// TIA Portal V17 export
// export: Created 2024-06-14T09:52:43.5267752Z, ExportSetting WithDefaults, DisplayName Totally Integrated Automation Portal, DisplayVersion V17, DisplayName TIA Portal Openness, DisplayVersion V17, DisplayName TIA Portal Version Control Interface, DisplayVersion V17, DisplayName Simotion SCOUT TIA, DisplayVersion 5.4.3.0, DisplayName SINAMICS Startdrive Advanced, DisplayVersion V17 SP1 Update 1, DisplayName SINAMICS Startdrive G110M, G120, G120C, G120D, G120P, G115D, DisplayVersion V17 SP1 Update 1, DisplayName SINAMICS Startdrive G130, G150, S120, S150, SINAMICS MV, S210, DisplayVersion V17 SP1 Update 1, DisplayName STEP 7 Professional, DisplayVersion V17, DisplayName STEP 7 Safety, DisplayVersion V17, DisplayName WinCC Professional, DisplayVersion V17
DATA_BLOCK "MOD_TCP_SETUP_DB"   // DB100
{ S7_Optimized_Access := 'FALSE' }
VERSION : 0.1
// stored: AutoNumber false, DBAccessibleFromOPCUA true, IsOnlyStoredInLoadMemory false, IsWriteProtectedInAS false
   VAR RETAIN
      TCP_Data_Station4 { ExternalAccessible := 'False'; ExternalVisible := 'False'; ExternalWritable := 'False'; S7_SetPoint := 'True'} : Array[1..6] of "Mod_TCP_Data";
      TCP_Data_Station5 { ExternalAccessible := 'False'; ExternalVisible := 'False'; ExternalWritable := 'False'} : Array[1..6] of "Mod_TCP_Data";
      TCP_Data_CHECK_SCALE_1 { S7_SetPoint := 'True'} : "Mod_TCP_Data";
      TCP_Data_CORRECTION_SCALE { S7_SetPoint := 'True'} : "Mod_TCP_Data";
   END_VAR
BEGIN
   TCP_Data_Station4[1..6].Mod_TCP_Connect.connectParamClient.InterfaceId := 64;
   TCP_Data_Station4[1].Mod_TCP_Connect.connectParamClient.ID := 1;
   TCP_Data_Station4[2].Mod_TCP_Connect.connectParamClient.ID := 2;
   TCP_Data_Station4[3].Mod_TCP_Connect.connectParamClient.ID := 3;
   TCP_Data_Station4[4].Mod_TCP_Connect.connectParamClient.ID := 4;
   TCP_Data_Station4[5].Mod_TCP_Connect.connectParamClient.ID := 5;
   TCP_Data_Station4[6].Mod_TCP_Connect.connectParamClient.ID := 6;
   TCP_Data_Station4[1..6].Mod_TCP_Connect.connectParamClient.ConnectionType := 16#0B;
   TCP_Data_Station4[1..6].Mod_TCP_Connect.connectParamClient.ActiveEstablished := true;
   TCP_Data_Station4[1].Mod_TCP_Connect.connectParamClient.RemoteAddress.ADDR[1] := 192;
   TCP_Data_Station4[1].Mod_TCP_Connect.connectParamClient.RemoteAddress.ADDR[2] := 168;
   TCP_Data_Station4[1].Mod_TCP_Connect.connectParamClient.RemoteAddress.ADDR[3] := 0;
   TCP_Data_Station4[1].Mod_TCP_Connect.connectParamClient.RemoteAddress.ADDR[4] := 21;
   TCP_Data_Station4[2].Mod_TCP_Connect.connectParamClient.RemoteAddress.ADDR[1] := 192;
   TCP_Data_Station4[2].Mod_TCP_Connect.connectParamClient.RemoteAddress.ADDR[2] := 168;
   TCP_Data_Station4[2].Mod_TCP_Connect.connectParamClient.RemoteAddress.ADDR[3] := 0;
   TCP_Data_Station4[2].Mod_TCP_Connect.connectParamClient.RemoteAddress.ADDR[4] := 22;
   TCP_Data_Station4[3].Mod_TCP_Connect.connectParamClient.RemoteAddress.ADDR[1] := 192;
   TCP_Data_Station4[3].Mod_TCP_Connect.connectParamClient.RemoteAddress.ADDR[2] := 168;
   TCP_Data_Station4[3].Mod_TCP_Connect.connectParamClient.RemoteAddress.ADDR[3] := 0;
   TCP_Data_Station4[3].Mod_TCP_Connect.connectParamClient.RemoteAddress.ADDR[4] := 23;
   TCP_Data_Station4[4].Mod_TCP_Connect.connectParamClient.RemoteAddress.ADDR[1] := 192;
   TCP_Data_Station4[4].Mod_TCP_Connect.connectParamClient.RemoteAddress.ADDR[2] := 168;
   TCP_Data_Station4[4].Mod_TCP_Connect.connectParamClient.RemoteAddress.ADDR[3] := 0;
   TCP_Data_Station4[4].Mod_TCP_Connect.connectParamClient.RemoteAddress.ADDR[4] := 24;
   TCP_Data_Station4[5].Mod_TCP_Connect.connectParamClient.RemoteAddress.ADDR[1] := 192;
   TCP_Data_Station4[5].Mod_TCP_Connect.connectParamClient.RemoteAddress.ADDR[2] := 168;
   TCP_Data_Station4[5].Mod_TCP_Connect.connectParamClient.RemoteAddress.ADDR[3] := 0;
   TCP_Data_Station4[5].Mod_TCP_Connect.connectParamClient.RemoteAddress.ADDR[4] := 25;
   TCP_Data_Station4[6].Mod_TCP_Connect.connectParamClient.RemoteAddress.ADDR[1] := 192;
   TCP_Data_Station4[6].Mod_TCP_Connect.connectParamClient.RemoteAddress.ADDR[2] := 168;
   TCP_Data_Station4[6].Mod_TCP_Connect.connectParamClient.RemoteAddress.ADDR[3] := 0;
   TCP_Data_Station4[6].Mod_TCP_Connect.connectParamClient.RemoteAddress.ADDR[4] := 26;
   TCP_Data_Station4[1..6].Mod_TCP_Connect.connectParamClient.RemotePort := 502;
   TCP_Data_Station4[2..6].Mod_TCP_Connect.connectParamClient.LocalPort := 0;
   TCP_Data_Station4[1].Mod_Client[1..6].request := false;
   TCP_Data_Station4[2].Mod_Client[1..6].request := false;
   TCP_Data_Station4[3].Mod_Client[1..6].request := false;
   TCP_Data_Station4[4].Mod_Client[1..6].request := false;
   TCP_Data_Station4[5].Mod_Client[1..6].request := false;
   TCP_Data_Station4[6].Mod_Client[1..6].request := false;
   TCP_Data_Station4[1].Mod_Client[1..6].enable := false;
   TCP_Data_Station4[2].Mod_Client[1..6].enable := false;
   TCP_Data_Station4[3].Mod_Client[1..6].enable := false;
   TCP_Data_Station4[4].Mod_Client[1..6].enable := false;
   TCP_Data_Station4[5].Mod_Client[1..6].enable := false;
   TCP_Data_Station4[6].Mod_Client[1..6].enable := false;
   TCP_Data_Station4[1].Mod_Client[1..6].disconnect := false;
   TCP_Data_Station4[2].Mod_Client[1..6].disconnect := false;
   TCP_Data_Station4[3].Mod_Client[1..6].disconnect := false;
   TCP_Data_Station4[4].Mod_Client[1..6].disconnect := false;
   TCP_Data_Station4[5].Mod_Client[1..6].disconnect := false;
   TCP_Data_Station4[6].Mod_Client[1..6].disconnect := false;
   TCP_Data_Station4[1].Mod_Client[1..6].done := false;
   TCP_Data_Station4[2].Mod_Client[1..6].done := false;
   TCP_Data_Station4[3].Mod_Client[1..6].done := false;
   TCP_Data_Station4[4].Mod_Client[1..6].done := false;
   TCP_Data_Station4[5].Mod_Client[1..6].done := false;
   TCP_Data_Station4[6].Mod_Client[1..6].done := false;
   TCP_Data_Station4[1].Mod_Client[1..6].busy := false;
   TCP_Data_Station4[2].Mod_Client[1..6].busy := false;
   TCP_Data_Station4[3].Mod_Client[1..6].busy := false;
   TCP_Data_Station4[4].Mod_Client[1..6].busy := false;
   TCP_Data_Station4[5].Mod_Client[1..6].busy := false;
   TCP_Data_Station4[6].Mod_Client[1..6].busy := false;
   TCP_Data_Station4[1].Mod_Client[1..6].error := false;
   TCP_Data_Station4[2].Mod_Client[1..6].error := false;
   TCP_Data_Station4[3].Mod_Client[1..6].error := false;
   TCP_Data_Station4[4].Mod_Client[1..6].error := false;
   TCP_Data_Station4[5].Mod_Client[1..6].error := false;
   TCP_Data_Station4[6].Mod_Client[1..6].error := false;
   TCP_Data_Station4[1].Mod_Client[1..6].status := 16#0;
   TCP_Data_Station4[2].Mod_Client[1..6].status := 16#0;
   TCP_Data_Station4[3].Mod_Client[1..6].status := 16#0;
   TCP_Data_Station4[4].Mod_Client[1..6].status := 16#0;
   TCP_Data_Station4[5].Mod_Client[1..6].status := 16#0;
   TCP_Data_Station4[6].Mod_Client[1..6].status := 16#0;
   TCP_Data_Station4[1].Mod_Client[1..6].statusSave := 16#0;
   TCP_Data_Station4[2].Mod_Client[1..6].statusSave := 16#0;
   TCP_Data_Station4[3].Mod_Client[1..6].statusSave := 16#0;
   TCP_Data_Station4[4].Mod_Client[1..6].statusSave := 16#0;
   TCP_Data_Station4[5].Mod_Client[1..6].statusSave := 16#0;
   TCP_Data_Station4[6].Mod_Client[1..6].statusSave := 16#0;
   TCP_Data_Station4[1].Mod_Client[1].modbusMode := 1;
   TCP_Data_Station4[1].Mod_Client[2].modbusMode := 0;
   TCP_Data_Station4[1].Mod_Client[3].modbusMode := 1;
   TCP_Data_Station4[1].Mod_Client[4..5].modbusMode := 0;
   TCP_Data_Station4[1].Mod_Client[6].modbusMode := 1;
   TCP_Data_Station4[2].Mod_Client[1].modbusMode := 1;
   TCP_Data_Station4[2].Mod_Client[2].modbusMode := 0;
   TCP_Data_Station4[2].Mod_Client[3].modbusMode := 1;
   TCP_Data_Station4[2].Mod_Client[4..5].modbusMode := 0;
   TCP_Data_Station4[2].Mod_Client[6].modbusMode := 1;
   TCP_Data_Station4[3].Mod_Client[1].modbusMode := 1;
   TCP_Data_Station4[3].Mod_Client[2].modbusMode := 0;
   TCP_Data_Station4[3].Mod_Client[3].modbusMode := 1;
   TCP_Data_Station4[3].Mod_Client[4..5].modbusMode := 0;
   TCP_Data_Station4[3].Mod_Client[6].modbusMode := 1;
   TCP_Data_Station4[4].Mod_Client[1].modbusMode := 1;
   TCP_Data_Station4[4].Mod_Client[2].modbusMode := 0;
   TCP_Data_Station4[4].Mod_Client[3].modbusMode := 1;
   TCP_Data_Station4[4].Mod_Client[4..5].modbusMode := 0;
   TCP_Data_Station4[4].Mod_Client[6].modbusMode := 1;
   TCP_Data_Station4[5].Mod_Client[1].modbusMode := 1;
   TCP_Data_Station4[5].Mod_Client[2].modbusMode := 0;
   TCP_Data_Station4[5].Mod_Client[3].modbusMode := 1;
   TCP_Data_Station4[5].Mod_Client[4..5].modbusMode := 0;
   TCP_Data_Station4[5].Mod_Client[6].modbusMode := 1;
   TCP_Data_Station4[6].Mod_Client[1].modbusMode := 1;
   TCP_Data_Station4[6].Mod_Client[2].modbusMode := 0;
   TCP_Data_Station4[6].Mod_Client[3].modbusMode := 1;
   TCP_Data_Station4[6].Mod_Client[4..5].modbusMode := 0;
   TCP_Data_Station4[6].Mod_Client[6].modbusMode := 1;
   TCP_Data_Station4[1].Mod_Client[1].modbusDataAddress := 40908;
   TCP_Data_Station4[1].Mod_Client[2].modbusDataAddress := 40001;
   TCP_Data_Station4[1].Mod_Client[3].modbusDataAddress := 40302;
   TCP_Data_Station4[1].Mod_Client[4].modbusDataAddress := 0;
   TCP_Data_Station4[1].Mod_Client[5].modbusDataAddress := 1;
   TCP_Data_Station4[1].Mod_Client[6].modbusDataAddress := 0;
   TCP_Data_Station4[2].Mod_Client[1].modbusDataAddress := 40908;
   TCP_Data_Station4[2].Mod_Client[2].modbusDataAddress := 40001;
   TCP_Data_Station4[2].Mod_Client[3].modbusDataAddress := 40302;
   TCP_Data_Station4[2].Mod_Client[4].modbusDataAddress := 0;
   TCP_Data_Station4[2].Mod_Client[5].modbusDataAddress := 1;
   TCP_Data_Station4[2].Mod_Client[6].modbusDataAddress := 0;
   TCP_Data_Station4[3].Mod_Client[1].modbusDataAddress := 40908;
   TCP_Data_Station4[3].Mod_Client[2].modbusDataAddress := 40001;
   TCP_Data_Station4[3].Mod_Client[3].modbusDataAddress := 40302;
   TCP_Data_Station4[3].Mod_Client[4].modbusDataAddress := 0;
   TCP_Data_Station4[3].Mod_Client[5].modbusDataAddress := 1;
   TCP_Data_Station4[3].Mod_Client[6].modbusDataAddress := 0;
   TCP_Data_Station4[4].Mod_Client[1].modbusDataAddress := 40908;
   TCP_Data_Station4[4].Mod_Client[2].modbusDataAddress := 40001;
   TCP_Data_Station4[4].Mod_Client[3].modbusDataAddress := 40302;
   TCP_Data_Station4[4].Mod_Client[4].modbusDataAddress := 0;
   TCP_Data_Station4[4].Mod_Client[5].modbusDataAddress := 1;
   TCP_Data_Station4[4].Mod_Client[6].modbusDataAddress := 0;
   TCP_Data_Station4[5].Mod_Client[1].modbusDataAddress := 40908;
   TCP_Data_Station4[5].Mod_Client[2].modbusDataAddress := 40001;
   TCP_Data_Station4[5].Mod_Client[3].modbusDataAddress := 40302;
   TCP_Data_Station4[5].Mod_Client[4].modbusDataAddress := 0;
   TCP_Data_Station4[5].Mod_Client[5].modbusDataAddress := 1;
   TCP_Data_Station4[5].Mod_Client[6].modbusDataAddress := 0;
   TCP_Data_Station4[6].Mod_Client[1].modbusDataAddress := 40908;
   TCP_Data_Station4[6].Mod_Client[2].modbusDataAddress := 40001;
   TCP_Data_Station4[6].Mod_Client[3].modbusDataAddress := 40302;
   TCP_Data_Station4[6].Mod_Client[4].modbusDataAddress := 0;
   TCP_Data_Station4[6].Mod_Client[5].modbusDataAddress := 1;
   TCP_Data_Station4[6].Mod_Client[6].modbusDataAddress := 0;
   TCP_Data_Station4[1].Mod_Client[1].modbusDataLen := 1;
   TCP_Data_Station4[1].Mod_Client[2].modbusDataLen := 6;
   TCP_Data_Station4[1].Mod_Client[3].modbusDataLen := 1;
   TCP_Data_Station4[1].Mod_Client[4].modbusDataLen := 0;
   TCP_Data_Station4[1].Mod_Client[5].modbusDataLen := 32;
   TCP_Data_Station4[1].Mod_Client[6].modbusDataLen := 1;
   TCP_Data_Station4[2].Mod_Client[1].modbusDataLen := 1;
   TCP_Data_Station4[2].Mod_Client[2].modbusDataLen := 6;
   TCP_Data_Station4[2].Mod_Client[3].modbusDataLen := 1;
   TCP_Data_Station4[2].Mod_Client[4].modbusDataLen := 0;
   TCP_Data_Station4[2].Mod_Client[5].modbusDataLen := 32;
   TCP_Data_Station4[2].Mod_Client[6].modbusDataLen := 1;
   TCP_Data_Station4[3].Mod_Client[1].modbusDataLen := 1;
   TCP_Data_Station4[3].Mod_Client[2].modbusDataLen := 6;
   TCP_Data_Station4[3].Mod_Client[3].modbusDataLen := 1;
   TCP_Data_Station4[3].Mod_Client[4].modbusDataLen := 0;
   TCP_Data_Station4[3].Mod_Client[5].modbusDataLen := 32;
   TCP_Data_Station4[3].Mod_Client[6].modbusDataLen := 1;
   TCP_Data_Station4[4].Mod_Client[1].modbusDataLen := 1;
   TCP_Data_Station4[4].Mod_Client[2].modbusDataLen := 6;
   TCP_Data_Station4[4].Mod_Client[3].modbusDataLen := 1;
   TCP_Data_Station4[4].Mod_Client[4].modbusDataLen := 0;
   TCP_Data_Station4[4].Mod_Client[5].modbusDataLen := 32;
   TCP_Data_Station4[4].Mod_Client[6].modbusDataLen := 1;
   TCP_Data_Station4[5].Mod_Client[1].modbusDataLen := 1;
   TCP_Data_Station4[5].Mod_Client[2].modbusDataLen := 6;
   TCP_Data_Station4[5].Mod_Client[3].modbusDataLen := 1;
   TCP_Data_Station4[5].Mod_Client[4].modbusDataLen := 0;
   TCP_Data_Station4[5].Mod_Client[5].modbusDataLen := 32;
   TCP_Data_Station4[5].Mod_Client[6].modbusDataLen := 1;
   TCP_Data_Station4[6].Mod_Client[1].modbusDataLen := 1;
   TCP_Data_Station4[6].Mod_Client[2].modbusDataLen := 6;
   TCP_Data_Station4[6].Mod_Client[3].modbusDataLen := 1;
   TCP_Data_Station4[6].Mod_Client[4].modbusDataLen := 0;
   TCP_Data_Station4[6].Mod_Client[5].modbusDataLen := 32;
   TCP_Data_Station4[6].Mod_Client[6].modbusDataLen := 1;
   TCP_Data_Station5[1..6].Mod_TCP_Connect.connectParamClient.InterfaceId := 64;
   TCP_Data_Station5[1].Mod_TCP_Connect.connectParamClient.ID := 11;
   TCP_Data_Station5[2].Mod_TCP_Connect.connectParamClient.ID := 12;
   TCP_Data_Station5[3].Mod_TCP_Connect.connectParamClient.ID := 13;
   TCP_Data_Station5[4].Mod_TCP_Connect.connectParamClient.ID := 14;
   TCP_Data_Station5[5].Mod_TCP_Connect.connectParamClient.ID := 15;
   TCP_Data_Station5[6].Mod_TCP_Connect.connectParamClient.ID := 16;
   TCP_Data_Station5[1..6].Mod_TCP_Connect.connectParamClient.ConnectionType := 16#0B;
   TCP_Data_Station5[1].Mod_TCP_Connect.connectParamClient.ActiveEstablished := true;
   TCP_Data_Station5[2..6].Mod_TCP_Connect.connectParamClient.ActiveEstablished := True;
   TCP_Data_Station5[1].Mod_TCP_Connect.connectParamClient.RemoteAddress.ADDR[1] := 192;
   TCP_Data_Station5[1].Mod_TCP_Connect.connectParamClient.RemoteAddress.ADDR[2] := 168;
   TCP_Data_Station5[1].Mod_TCP_Connect.connectParamClient.RemoteAddress.ADDR[3] := 0;
   TCP_Data_Station5[1].Mod_TCP_Connect.connectParamClient.RemoteAddress.ADDR[4] := 31;
   TCP_Data_Station5[2].Mod_TCP_Connect.connectParamClient.RemoteAddress.ADDR[1] := 192;
   TCP_Data_Station5[2].Mod_TCP_Connect.connectParamClient.RemoteAddress.ADDR[2] := 168;
   TCP_Data_Station5[2].Mod_TCP_Connect.connectParamClient.RemoteAddress.ADDR[3] := 0;
   TCP_Data_Station5[2].Mod_TCP_Connect.connectParamClient.RemoteAddress.ADDR[4] := 32;
   TCP_Data_Station5[3].Mod_TCP_Connect.connectParamClient.RemoteAddress.ADDR[1] := 192;
   TCP_Data_Station5[3].Mod_TCP_Connect.connectParamClient.RemoteAddress.ADDR[2] := 168;
   TCP_Data_Station5[3].Mod_TCP_Connect.connectParamClient.RemoteAddress.ADDR[3] := 0;
   TCP_Data_Station5[3].Mod_TCP_Connect.connectParamClient.RemoteAddress.ADDR[4] := 33;
   TCP_Data_Station5[4].Mod_TCP_Connect.connectParamClient.RemoteAddress.ADDR[1] := 192;
   TCP_Data_Station5[4].Mod_TCP_Connect.connectParamClient.RemoteAddress.ADDR[2] := 168;
   TCP_Data_Station5[4].Mod_TCP_Connect.connectParamClient.RemoteAddress.ADDR[3] := 0;
   TCP_Data_Station5[4].Mod_TCP_Connect.connectParamClient.RemoteAddress.ADDR[4] := 34;
   TCP_Data_Station5[5].Mod_TCP_Connect.connectParamClient.RemoteAddress.ADDR[1] := 192;
   TCP_Data_Station5[5].Mod_TCP_Connect.connectParamClient.RemoteAddress.ADDR[2] := 168;
   TCP_Data_Station5[5].Mod_TCP_Connect.connectParamClient.RemoteAddress.ADDR[3] := 0;
   TCP_Data_Station5[5].Mod_TCP_Connect.connectParamClient.RemoteAddress.ADDR[4] := 35;
   TCP_Data_Station5[6].Mod_TCP_Connect.connectParamClient.RemoteAddress.ADDR[1] := 192;
   TCP_Data_Station5[6].Mod_TCP_Connect.connectParamClient.RemoteAddress.ADDR[2] := 168;
   TCP_Data_Station5[6].Mod_TCP_Connect.connectParamClient.RemoteAddress.ADDR[3] := 0;
   TCP_Data_Station5[6].Mod_TCP_Connect.connectParamClient.RemoteAddress.ADDR[4] := 36;
   TCP_Data_Station5[1..6].Mod_TCP_Connect.connectParamClient.RemotePort := 502;
   TCP_Data_Station5[1..6].Mod_TCP_Connect.connectParamClient.LocalPort := 0;
   TCP_Data_Station5[1].Mod_Client[1..6].request := false;
   TCP_Data_Station5[2].Mod_Client[1..6].request := false;
   TCP_Data_Station5[3].Mod_Client[1..6].request := false;
   TCP_Data_Station5[4].Mod_Client[1..6].request := false;
   TCP_Data_Station5[5].Mod_Client[1..6].request := false;
   TCP_Data_Station5[6].Mod_Client[1..6].request := false;
   TCP_Data_Station5[1].Mod_Client[1..6].enable := false;
   TCP_Data_Station5[2].Mod_Client[1..6].enable := false;
   TCP_Data_Station5[3].Mod_Client[1..6].enable := false;
   TCP_Data_Station5[4].Mod_Client[1..6].enable := false;
   TCP_Data_Station5[5].Mod_Client[1..6].enable := false;
   TCP_Data_Station5[6].Mod_Client[1..6].enable := false;
   TCP_Data_Station5[1].Mod_Client[1..6].disconnect := false;
   TCP_Data_Station5[2].Mod_Client[1..6].disconnect := false;
   TCP_Data_Station5[3].Mod_Client[1..6].disconnect := false;
   TCP_Data_Station5[4].Mod_Client[1..6].disconnect := false;
   TCP_Data_Station5[5].Mod_Client[1..6].disconnect := false;
   TCP_Data_Station5[6].Mod_Client[1..6].disconnect := false;
   TCP_Data_Station5[1].Mod_Client[1..6].done := false;
   TCP_Data_Station5[2].Mod_Client[1..6].done := false;
   TCP_Data_Station5[3].Mod_Client[1..6].done := false;
   TCP_Data_Station5[4].Mod_Client[1..6].done := false;
   TCP_Data_Station5[5].Mod_Client[1..6].done := false;
   TCP_Data_Station5[6].Mod_Client[1..6].done := false;
   TCP_Data_Station5[1].Mod_Client[1..6].busy := false;
   TCP_Data_Station5[2].Mod_Client[1..6].busy := false;
   TCP_Data_Station5[3].Mod_Client[1..6].busy := false;
   TCP_Data_Station5[4].Mod_Client[1..6].busy := false;
   TCP_Data_Station5[5].Mod_Client[1..6].busy := false;
   TCP_Data_Station5[6].Mod_Client[1..6].busy := false;
   TCP_Data_Station5[1].Mod_Client[1..6].error := false;
   TCP_Data_Station5[2].Mod_Client[1..6].error := false;
   TCP_Data_Station5[3].Mod_Client[1..6].error := false;
   TCP_Data_Station5[4].Mod_Client[1..6].error := false;
   TCP_Data_Station5[5].Mod_Client[1..6].error := false;
   TCP_Data_Station5[6].Mod_Client[1..6].error := false;
   TCP_Data_Station5[1].Mod_Client[1..6].status := 16#0;
   TCP_Data_Station5[2].Mod_Client[1..6].status := 16#0;
   TCP_Data_Station5[3].Mod_Client[1..6].status := 16#0;
   TCP_Data_Station5[4].Mod_Client[1..6].status := 16#0;
   TCP_Data_Station5[5].Mod_Client[1..6].status := 16#0;
   TCP_Data_Station5[6].Mod_Client[1..6].status := 16#0;
   TCP_Data_Station5[1].Mod_Client[1..6].statusSave := 16#0;
   TCP_Data_Station5[2].Mod_Client[1..6].statusSave := 16#0;
   TCP_Data_Station5[3].Mod_Client[1..6].statusSave := 16#0;
   TCP_Data_Station5[4].Mod_Client[1..6].statusSave := 16#0;
   TCP_Data_Station5[5].Mod_Client[1..6].statusSave := 16#0;
   TCP_Data_Station5[6].Mod_Client[1..6].statusSave := 16#0;
   TCP_Data_Station5[1].Mod_Client[1].modbusMode := 1;
   TCP_Data_Station5[1].Mod_Client[2].modbusMode := 0;
   TCP_Data_Station5[1].Mod_Client[3].modbusMode := 1;
   TCP_Data_Station5[1].Mod_Client[4..5].modbusMode := 0;
   TCP_Data_Station5[1].Mod_Client[6].modbusMode := 1;
   TCP_Data_Station5[2].Mod_Client[1].modbusMode := 1;
   TCP_Data_Station5[2].Mod_Client[2].modbusMode := 0;
   TCP_Data_Station5[2].Mod_Client[3].modbusMode := 1;
   TCP_Data_Station5[2].Mod_Client[4..5].modbusMode := 0;
   TCP_Data_Station5[2].Mod_Client[6].modbusMode := 1;
   TCP_Data_Station5[3].Mod_Client[1].modbusMode := 1;
   TCP_Data_Station5[3].Mod_Client[2].modbusMode := 0;
   TCP_Data_Station5[3].Mod_Client[3].modbusMode := 1;
   TCP_Data_Station5[3].Mod_Client[4..5].modbusMode := 0;
   TCP_Data_Station5[3].Mod_Client[6].modbusMode := 1;
   TCP_Data_Station5[4].Mod_Client[1].modbusMode := 1;
   TCP_Data_Station5[4].Mod_Client[2].modbusMode := 0;
   TCP_Data_Station5[4].Mod_Client[3].modbusMode := 1;
   TCP_Data_Station5[4].Mod_Client[4..5].modbusMode := 0;
   TCP_Data_Station5[4].Mod_Client[6].modbusMode := 1;
   TCP_Data_Station5[5].Mod_Client[1].modbusMode := 1;
   TCP_Data_Station5[5].Mod_Client[2].modbusMode := 0;
   TCP_Data_Station5[5].Mod_Client[3].modbusMode := 1;
   TCP_Data_Station5[5].Mod_Client[4..5].modbusMode := 0;
   TCP_Data_Station5[5].Mod_Client[6].modbusMode := 1;
   TCP_Data_Station5[6].Mod_Client[1].modbusMode := 1;
   TCP_Data_Station5[6].Mod_Client[2].modbusMode := 0;
   TCP_Data_Station5[6].Mod_Client[3].modbusMode := 1;
   TCP_Data_Station5[6].Mod_Client[4..5].modbusMode := 0;
   TCP_Data_Station5[6].Mod_Client[6].modbusMode := 1;
   TCP_Data_Station5[1].Mod_Client[1].modbusDataAddress := 40908;
   TCP_Data_Station5[1].Mod_Client[2].modbusDataAddress := 40001;
   TCP_Data_Station5[1].Mod_Client[3].modbusDataAddress := 40302;
   TCP_Data_Station5[1].Mod_Client[4].modbusDataAddress := 0;
   TCP_Data_Station5[1].Mod_Client[5].modbusDataAddress := 1;
   TCP_Data_Station5[1].Mod_Client[6].modbusDataAddress := 0;
   TCP_Data_Station5[2].Mod_Client[1].modbusDataAddress := 40908;
   TCP_Data_Station5[2].Mod_Client[2].modbusDataAddress := 40001;
   TCP_Data_Station5[2].Mod_Client[3].modbusDataAddress := 40302;
   TCP_Data_Station5[2].Mod_Client[4].modbusDataAddress := 0;
   TCP_Data_Station5[2].Mod_Client[5].modbusDataAddress := 1;
   TCP_Data_Station5[2].Mod_Client[6].modbusDataAddress := 0;
   TCP_Data_Station5[3].Mod_Client[1].modbusDataAddress := 40908;
   TCP_Data_Station5[3].Mod_Client[2].modbusDataAddress := 40001;
   TCP_Data_Station5[3].Mod_Client[3].modbusDataAddress := 40302;
   TCP_Data_Station5[3].Mod_Client[4].modbusDataAddress := 0;
   TCP_Data_Station5[3].Mod_Client[5].modbusDataAddress := 1;
   TCP_Data_Station5[3].Mod_Client[6].modbusDataAddress := 0;
   TCP_Data_Station5[4].Mod_Client[1].modbusDataAddress := 40908;
   TCP_Data_Station5[4].Mod_Client[2].modbusDataAddress := 40001;
   TCP_Data_Station5[4].Mod_Client[3].modbusDataAddress := 40302;
   TCP_Data_Station5[4].Mod_Client[4].modbusDataAddress := 0;
   TCP_Data_Station5[4].Mod_Client[5].modbusDataAddress := 1;
   TCP_Data_Station5[4].Mod_Client[6].modbusDataAddress := 0;
   TCP_Data_Station5[5].Mod_Client[1].modbusDataAddress := 40908;
   TCP_Data_Station5[5].Mod_Client[2].modbusDataAddress := 40001;
   TCP_Data_Station5[5].Mod_Client[3].modbusDataAddress := 40302;
   TCP_Data_Station5[5].Mod_Client[4].modbusDataAddress := 0;
   TCP_Data_Station5[5].Mod_Client[5].modbusDataAddress := 1;
   TCP_Data_Station5[5].Mod_Client[6].modbusDataAddress := 0;
   TCP_Data_Station5[6].Mod_Client[1].modbusDataAddress := 40908;
   TCP_Data_Station5[6].Mod_Client[2].modbusDataAddress := 40001;
   TCP_Data_Station5[6].Mod_Client[3].modbusDataAddress := 40302;
   TCP_Data_Station5[6].Mod_Client[4].modbusDataAddress := 0;
   TCP_Data_Station5[6].Mod_Client[5].modbusDataAddress := 1;
   TCP_Data_Station5[6].Mod_Client[6].modbusDataAddress := 0;
   TCP_Data_Station5[1].Mod_Client[1].modbusDataLen := 1;
   TCP_Data_Station5[1].Mod_Client[2].modbusDataLen := 6;
   TCP_Data_Station5[1].Mod_Client[3].modbusDataLen := 1;
   TCP_Data_Station5[1].Mod_Client[4].modbusDataLen := 0;
   TCP_Data_Station5[1].Mod_Client[5].modbusDataLen := 32;
   TCP_Data_Station5[1].Mod_Client[6].modbusDataLen := 1;
   TCP_Data_Station5[2].Mod_Client[1].modbusDataLen := 1;
   TCP_Data_Station5[2].Mod_Client[2].modbusDataLen := 6;
   TCP_Data_Station5[2].Mod_Client[3].modbusDataLen := 1;
   TCP_Data_Station5[2].Mod_Client[4].modbusDataLen := 0;
   TCP_Data_Station5[2].Mod_Client[5].modbusDataLen := 32;
   TCP_Data_Station5[2].Mod_Client[6].modbusDataLen := 1;
   TCP_Data_Station5[3].Mod_Client[1].modbusDataLen := 1;
   TCP_Data_Station5[3].Mod_Client[2].modbusDataLen := 6;
   TCP_Data_Station5[3].Mod_Client[3].modbusDataLen := 1;
   TCP_Data_Station5[3].Mod_Client[4].modbusDataLen := 0;
   TCP_Data_Station5[3].Mod_Client[5].modbusDataLen := 32;
   TCP_Data_Station5[3].Mod_Client[6].modbusDataLen := 1;
   TCP_Data_Station5[4].Mod_Client[1].modbusDataLen := 1;
   TCP_Data_Station5[4].Mod_Client[2].modbusDataLen := 6;
   TCP_Data_Station5[4].Mod_Client[3].modbusDataLen := 1;
   TCP_Data_Station5[4].Mod_Client[4].modbusDataLen := 0;
   TCP_Data_Station5[4].Mod_Client[5].modbusDataLen := 32;
   TCP_Data_Station5[4].Mod_Client[6].modbusDataLen := 1;
   TCP_Data_Station5[5].Mod_Client[1].modbusDataLen := 1;
   TCP_Data_Station5[5].Mod_Client[2].modbusDataLen := 6;
   TCP_Data_Station5[5].Mod_Client[3].modbusDataLen := 1;
   TCP_Data_Station5[5].Mod_Client[4].modbusDataLen := 0;
   TCP_Data_Station5[5].Mod_Client[5].modbusDataLen := 32;
   TCP_Data_Station5[5].Mod_Client[6].modbusDataLen := 1;
   TCP_Data_Station5[6].Mod_Client[1].modbusDataLen := 1;
   TCP_Data_Station5[6].Mod_Client[2].modbusDataLen := 6;
   TCP_Data_Station5[6].Mod_Client[3].modbusDataLen := 1;
   TCP_Data_Station5[6].Mod_Client[4].modbusDataLen := 0;
   TCP_Data_Station5[6].Mod_Client[5].modbusDataLen := 32;
   TCP_Data_Station5[6].Mod_Client[6].modbusDataLen := 1;
   TCP_Data_CHECK_SCALE_1.Mod_TCP_Connect.connectParamClient.InterfaceId := 64;
   TCP_Data_CHECK_SCALE_1.Mod_TCP_Connect.connectParamClient.ID := 21;
   TCP_Data_CHECK_SCALE_1.Mod_TCP_Connect.connectParamClient.ConnectionType := 16#0B;
   TCP_Data_CHECK_SCALE_1.Mod_TCP_Connect.connectParamClient.ActiveEstablished := true;
   TCP_Data_CHECK_SCALE_1.Mod_TCP_Connect.connectParamClient.RemoteAddress.ADDR[1] := 192;
   TCP_Data_CHECK_SCALE_1.Mod_TCP_Connect.connectParamClient.RemoteAddress.ADDR[2] := 168;
   TCP_Data_CHECK_SCALE_1.Mod_TCP_Connect.connectParamClient.RemoteAddress.ADDR[3] := 0;
   TCP_Data_CHECK_SCALE_1.Mod_TCP_Connect.connectParamClient.RemoteAddress.ADDR[4] := 41;
   TCP_Data_CHECK_SCALE_1.Mod_TCP_Connect.connectParamClient.RemotePort := 502;
   TCP_Data_CHECK_SCALE_1.Mod_TCP_Connect.connectParamClient.LocalPort := 0;
   TCP_Data_CHECK_SCALE_1.Mod_Client[1..6].request := false;
   TCP_Data_CHECK_SCALE_1.Mod_Client[1..6].enable := false;
   TCP_Data_CHECK_SCALE_1.Mod_Client[1..6].disconnect := false;
   TCP_Data_CHECK_SCALE_1.Mod_Client[1..6].done := false;
   TCP_Data_CHECK_SCALE_1.Mod_Client[1..6].busy := false;
   TCP_Data_CHECK_SCALE_1.Mod_Client[1..6].error := false;
   TCP_Data_CHECK_SCALE_1.Mod_Client[1..6].status := 16#0;
   TCP_Data_CHECK_SCALE_1.Mod_Client[1..6].statusSave := 16#0;
   TCP_Data_CHECK_SCALE_1.Mod_Client[1].modbusMode := 1;
   TCP_Data_CHECK_SCALE_1.Mod_Client[2].modbusMode := 0;
   TCP_Data_CHECK_SCALE_1.Mod_Client[3].modbusMode := 1;
   TCP_Data_CHECK_SCALE_1.Mod_Client[4..5].modbusMode := 0;
   TCP_Data_CHECK_SCALE_1.Mod_Client[6].modbusMode := 1;
   TCP_Data_CHECK_SCALE_1.Mod_Client[1].modbusDataAddress := 40908;
   TCP_Data_CHECK_SCALE_1.Mod_Client[2].modbusDataAddress := 40011;
   TCP_Data_CHECK_SCALE_1.Mod_Client[3].modbusDataAddress := 40302;
   TCP_Data_CHECK_SCALE_1.Mod_Client[4].modbusDataAddress := 0;
   TCP_Data_CHECK_SCALE_1.Mod_Client[5].modbusDataAddress := 1;
   TCP_Data_CHECK_SCALE_1.Mod_Client[6].modbusDataAddress := 0;
   TCP_Data_CHECK_SCALE_1.Mod_Client[1].modbusDataLen := 1;
   TCP_Data_CHECK_SCALE_1.Mod_Client[2].modbusDataLen := 10;
   TCP_Data_CHECK_SCALE_1.Mod_Client[3].modbusDataLen := 1;
   TCP_Data_CHECK_SCALE_1.Mod_Client[4].modbusDataLen := 0;
   TCP_Data_CHECK_SCALE_1.Mod_Client[5].modbusDataLen := 32;
   TCP_Data_CHECK_SCALE_1.Mod_Client[6].modbusDataLen := 1;
   TCP_Data_CORRECTION_SCALE.Mod_TCP_Connect.connectParamClient.InterfaceId := 64;
   TCP_Data_CORRECTION_SCALE.Mod_TCP_Connect.connectParamClient.ID := 41;
   TCP_Data_CORRECTION_SCALE.Mod_TCP_Connect.connectParamClient.ConnectionType := 16#0B;
   TCP_Data_CORRECTION_SCALE.Mod_TCP_Connect.connectParamClient.ActiveEstablished := TRUE;
   TCP_Data_CORRECTION_SCALE.Mod_TCP_Connect.connectParamClient.RemoteAddress.ADDR[1] := 192;
   TCP_Data_CORRECTION_SCALE.Mod_TCP_Connect.connectParamClient.RemoteAddress.ADDR[2] := 168;
   TCP_Data_CORRECTION_SCALE.Mod_TCP_Connect.connectParamClient.RemoteAddress.ADDR[3] := 0;
   TCP_Data_CORRECTION_SCALE.Mod_TCP_Connect.connectParamClient.RemoteAddress.ADDR[4] := 41;
   TCP_Data_CORRECTION_SCALE.Mod_TCP_Connect.connectParamClient.RemotePort := 502;
END_DATA_BLOCK
